# EPICS substitutions: current/app/Db/ValveOutputs.substitutions
file hpm900mbbiDirect.template {
  pattern {RECORD_NAME, OFFSET, FANOUT_RECORD}
  {VALVE_OUTPUTS_RBV, 40, VALVE_OUTPUTS_FANOUT}
}

file fanout12bit.template {
    pattern {RECORD_NAME,LINK0,LINK1,LINK2,LINK3,LINK4,LINK5,LINK6,LINK7,LINK8,LINK9,LINKA,LINKB}
    {VALVE_OUTPUTS_FANOUT,
     LPI:2:OPN_DO_RBV,
     LPV:2:OPN_DO_RBV,
     VGS:2:OPN_DO_RBV,
     HPV:2:OPN_DO_RBV,
     HPI:2:OPN_DO_RBV,
     PGI:2:OPN_DO_RBV,
     LPI:1:OPN_DO_RBV,
     LPV:1:OPN_DO_RBV,
     VGS:1:OPN_DO_RBV,
     HPV:1:OPN_DO_RBV,
     HPI:1:OPN_DO_RBV,
     PGI:1:OPN_DO_RBV}
}

file hpm900bi.template {
    pattern {RECORD_NAME, DESC, BIT, INP}
    {HPI:2:OPN_DO_RBV, "HPI 2 valve position state", 0, VALVE_OUTPUTS_RBV}
    {HPV:2:OPN_DO_RBV, "HPV 2 valve position state", 1, VALVE_OUTPUTS_RBV}
    {PGI:2:OPN_DO_RBV, "PGI 2 valve position state", 2, VALVE_OUTPUTS_RBV}
    {LPI:2:OPN_DO_RBV, "LPI 2 valve position state", 3, VALVE_OUTPUTS_RBV}
    {LPV:2:OPN_DO_RBV, "LPV 2 valve position state", 4, VALVE_OUTPUTS_RBV}
    {VGS:2:OPN_DO_RBV, "VGS 2 valve position state", 5, VALVE_OUTPUTS_RBV}
    {HPI:1:OPN_DO_RBV, "HPI 1 valve position state", 8, VALVE_OUTPUTS_RBV}
    {HPV:1:OPN_DO_RBV, "HPV 1 valve position state", 9, VALVE_OUTPUTS_RBV}
    {PGI:1:OPN_DO_RBV, "PGI 1 valve position state", A, VALVE_OUTPUTS_RBV}
    {LPI:1:OPN_DO_RBV, "LPI 1 valve position state", B, VALVE_OUTPUTS_RBV}
    {LPV:1:OPN_DO_RBV, "LPV 1 valve position state", C, VALVE_OUTPUTS_RBV}
    {VGS:1:OPN_DO_RBV, "VGS 1 valve position state", D, VALVE_OUTPUTS_RBV}
}
